// TIA Portal V21 export
FUNCTION_BLOCK "BatchDetailsLength"   // FB99, LAD
{ S7_Optimized_Access := 'TRUE' }
// stored: AutoNumber false, MemoryReserve 100, SetENOAutomatically false
   VAR_OUTPUT
      EquipmentID_Len { ExternalAccessible := 'False'; ExternalVisible := 'False'; ExternalWritable := 'False'} : Int;
      ProductName_Len { ExternalAccessible := 'False'; ExternalVisible := 'False'; ExternalWritable := 'False'} : Int;
      BatchNum_Len { ExternalAccessible := 'False'; ExternalVisible := 'False'; ExternalWritable := 'False'} : Int;
      PrintInt_Len { ExternalAccessible := 'False'; ExternalVisible := 'False'; ExternalWritable := 'False'} : Int;
   END_VAR
   VAR_TEMP   // added for the SCL form of the ladder/FBD networks
      _w1 : Bool;
      _w2 : Bool;
   END_VAR
BEGIN

REGION Network 1: BATCH DETAIL LENGTH
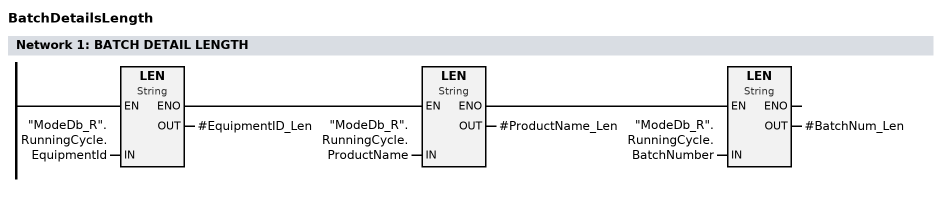
   RUNG wire#powerrail
      { S7_Templates := "[str_type := String, return_type := Int]" } LEN(IN := "ModeDb_R".RunningCycle.EquipmentId, OUT => #EquipmentID_Len)
      { S7_Templates := "[str_type := String, return_type := Int]" } LEN(IN := "ModeDb_R".RunningCycle.ProductName, OUT => #ProductName_Len)
      { S7_Templates := "[str_type := String, return_type := Int]" } LEN(IN := "ModeDb_R".RunningCycle.BatchNumber, OUT => #BatchNum_Len)
   END_RUNG
   // the same network as SCL:
   LEN(IN := "ModeDb_R".RunningCycle.EquipmentId, OUT => #EquipmentID_Len, ENO => #_w1);
   LEN(EN := #_w1, IN := "ModeDb_R".RunningCycle.ProductName, OUT => #ProductName_Len, ENO => #_w2);
   IF #_w2 THEN LEN(IN := "ModeDb_R".RunningCycle.BatchNumber, OUT => #BatchNum_Len); END_IF;
END_REGION
END_FUNCTION_BLOCK
